{attribute 'linkalways'} 
{attribute 'no_explicit_call' := 'This FB is a CLASS and must be accessed using methods or properties'}
{attribute 'enable_dynamic_creation'}
FUNCTION_BLOCK FINAL AND_DWORD EXTENDS Node
VAR
	in1 : _DWORD(0);
	in2 : _DWORD(0);
	out : _DWORD(0);
END_VAR

METHOD PUBLIC Clone : I_Node
VAR
	pNode : POINTER TO AND_DWORD;
END_VAR
pNode := __NEW(AND_DWORD);
Clone := pNode^;
END_METHOD

METHOD FB_init : BOOL
VAR_INPUT
	bInitRetains : BOOL; // if TRUE, the retain variables are initialized (warm start / cold start)
	bInCopyCode : BOOL;  // if TRUE, the instance afterwards gets moved into the copy code (online change)
END_VAR
AddInput('in1',THIS^.in1);
AddInput('in2',THIS^.in2);
AddOutput('out', THIS^.out);
END_METHOD

METHOD PROTECTED OnExecute
VAR
END_VAR
out.Value := in1.Value AND in2.Value;
END_METHOD

END_FUNCTION_BLOCK

(* stored: Version 1.1.0.1, ProductVersion 3.1.4024.15
   POU AND_DWORD: Id {4eafe7f6-81c3-41c4-b794-db11738388ce}, SpecialFunc None
   Folder Constructor: Id {0c735dd9-1d0f-4ab1-b7ed-5d81017b5bfc}
   Method Clone: Id {cf88f5b3-5481-4069-af1b-7dc640527bad}
   Method FB_init: Id {f5ea8dbb-b7f1-4df3-9ab8-c7acfd8bd63f}
   Method OnExecute: Id {e3b0b3eb-43b0-41fc-9d1e-654eb45f0277} *)
